Staubli VAL3: start.pgx

program start()
begin
  // Initialisation
  call init()

  // Creation tache suivi position toutes les 4ms
  taskCreateSync sTaskPos, 0.004, bOvrPosition, tPosition()

  // On attend qu'elle soit démarree
  wait(taskStatus(sTaskPos)==1)



  // Lancement du process principal
  taskCreate sTaskRobot, 100, tRobot()
  wait(taskStatus(sTaskRobot)==1)

  // Surveillance
  while true
    if nPrevOvrPos!=nOvrPos
      logMsg("Overrun dans la tache "+sTaskPos)
      nPrevOvrPos=nOvrPos
    endIf

    delay(0)
  endWhile
end
